// TIA Portal V18 export
DATA_BLOCK "EPICSData"   // DB8
{ S7_Optimized_Access := 'FALSE'; DB_Accessible_From_OPC_UA := 'FALSE' }
VERSION : 0.1
// stored: AutoNumber true, DBAccessibleFromOPCUA false, IsOnlyStoredInLoadMemory false, IsWriteProtectedInAS false
   VAR
      Reset : Bool;
   END_VAR
BEGIN
END_DATA_BLOCK
